// Mitsubishi GX Works2 project: main_plus   PLC: Q02/Q02H

PROGRAM MAIN
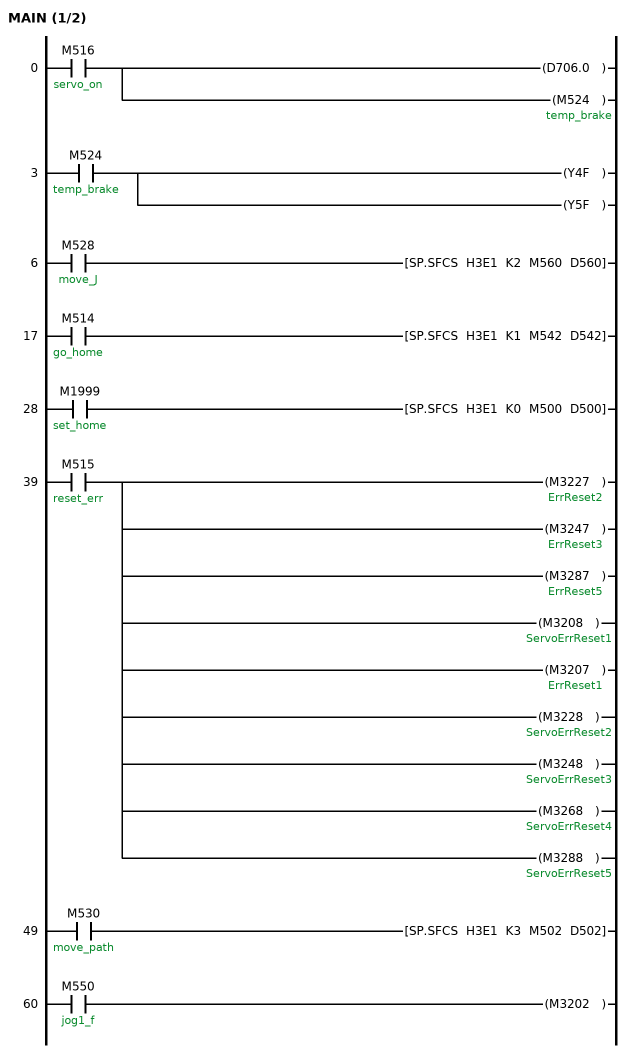
0     LD      M516  ; servo_on
      OUT     D706.0
      OUT     M524  ; temp_brake
3     LD      M524  ; temp_brake
      OUT     Y4F
      OUT     Y5F
6     LD      M528  ; move_J
      SP.SFCS H3E1 K2 M560 D560
17    LD      M514  ; go_home
      SP.SFCS H3E1 K1 M542 D542
28    LD      M1999  ; set_home
      SP.SFCS H3E1 K0 M500 D500
39    LD      M515  ; reset_err
      OUT     M3227  ; ErrReset2
      OUT     M3247  ; ErrReset3
      OUT     M3287  ; ErrReset5
      OUT     M3208  ; ServoErrReset1
      OUT     M3207  ; ErrReset1
      OUT     M3228  ; ServoErrReset2
      OUT     M3248  ; ServoErrReset3
      OUT     M3268  ; ServoErrReset4
      OUT     M3288  ; ServoErrReset5
49    LD      M530  ; move_path
      SP.SFCS H3E1 K3 M502 D502
60    LD      M550  ; jog1_f
      OUT     M3202
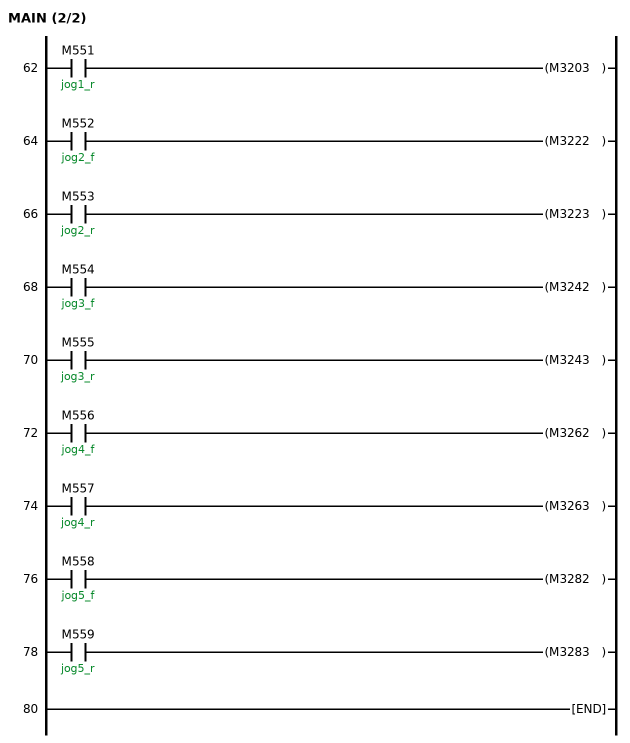
62    LD      M551  ; jog1_r
      OUT     M3203
64    LD      M552  ; jog2_f
      OUT     M3222
66    LD      M553  ; jog2_r
      OUT     M3223
68    LD      M554  ; jog3_f
      OUT     M3242
70    LD      M555  ; jog3_r
      OUT     M3243
72    LD      M556  ; jog4_f
      OUT     M3262
74    LD      M557  ; jog4_r
      OUT     M3263
76    LD      M558  ; jog5_f
      OUT     M3282
78    LD      M559  ; jog5_r
      OUT     M3283
80    END
END_PROGRAM

// device comments not shown above
D0  ; FeedCVal1
D20  ; FeedCVal2
D40  ; FeedCVal3
D60  ; FeedCVal4
D80  ; FeedCVal5
D704  ; PLC ready flag request
D705  ; passpoint
D706  ; on_servo
D858  ; getpoint
D859  ; run
D1010  ; start_100_point
D1012  ; theta2
D1014  ; theta3
D1016  ; theta4
D1018  ; theta5
D2000  ; v1
D2002  ; v2
D2004  ; v3
D2006  ; v4
D2008  ; v5
D2010  ; addresspoint1
D2012  ; addresspoint2
D2014  ; addresspoint3
D2016  ; addresspoint4
D2018  ; addresspoint5
D10302  ; No.Protocol
D10320  ; slaveID
D10321  ; address
D10322  ; No.Resister
M154  ; go_home
M512  ; PLC ready flag request
M513  ; brake
M543  ; position
M544  ; speed
M590  ; move_path2
M1000  ; Accep flag 1
M1001  ; Accep flag 2
M1002  ; Accep flag 3
M1003  ; Accep flag 4
M1004  ; Accep flag 5
M1005  ; Servo ready 1
M1006  ; Servo ready 2
M1007  ; Servo ready 3
M1008  ; Servo ready 4
M1009  ; Servo ready 5
M1010  ; Error 1
M1011  ; Error 2
M1012  ; Error 3
M1013  ; Error 4
M1014  ; Error 5
M1015  ; ready flag
M1016  ; brake
M1987  ; reset
M1988  ; conveyor
M1989  ; symetric
M1993  ; manrun
M1994  ; modbus
M1995  ; runall
M1996  ; getpoint
M1997  ; moveJog
M1998  ; ReHome
M2000  ; PLC Ready flag
M2001  ; StartAceptFlag1
M2002  ; StartAceptFlag2
M2003  ; StartAceptFlag3
M2004  ; StartAceptFlag4
M2005  ; StartAceptFlag5
M2407  ; ErrDetec1
M2408  ; SerErrDetec1
M2415  ; ServoReady1
M2427  ; ErrDetec2
M2428  ; SerErrDetec2
M2435  ; ServoReady2
M2447  ; ErrDetec3
M2448  ; SerErrDetec3
M2455  ; ServoReady3
M2467  ; ErrDetec4
M2468  ; SerErrDetec4
M2475  ; ServoReady4
M2487  ; ErrDetec5
M2488  ; SerErrDetec5
M2495  ; ServoReady5
M3000  ; brake_2
M3010  ; brak_3
M3020  ; xylanh
M3030  ; on_servo
M3267  ; ErrReset4
M3840  ; SFC flag
M3842  ; get camera
M3843  ; Run Only
M3844  ; gang tay
T0  ; timer out
